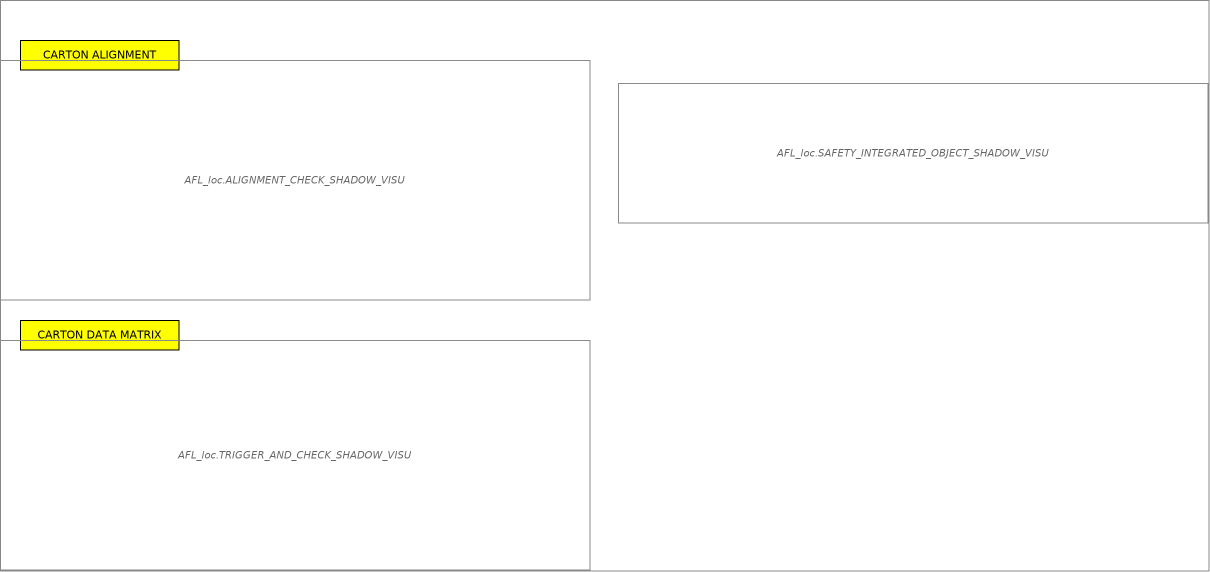
VISUALIZATION CARTON_FORMING_CHECKS  // 1210x572
    Rectangle (20,40 159x30), "CARTON ALIGNMENT"
    Frame (0,60 590x240)
        shows AFL_loc.ALIGNMENT_CHECK_SHADOW_VISU(m_Input_alignment_check_shadow := dbg_wu_cartonforming_belt_checks.algnchk_shd)
    Rectangle (20,320 159x30), "CARTON DATA MATRIX"
    Frame (0,340 590x230)
        shows AFL_loc.TRIGGER_AND_CHECK_SHADOW_VISU(m_Input_trigger_and_check_shadow := dbg_wu_cartonforming_belt_checks.data_matrix_tchk_shd)
    Frame (618,83 590x140)
        shows AFL_loc.SAFETY_INTEGRATED_OBJECT_SHADOW_VISU(m_Input_safety_integrated_object_shadow := dbg_wu_main_safety_guards.sio_shd)
END_VISUALIZATION

(* stored: Version 1.1.0.1, ProductVersion 3.1.4024.3
   Visu CARTON_FORMING_CHECKS: Id {41b6774d-e0bd-4eb6-8d93-d57638868a57} *)
